TYPE AC_Unit_Status :
STRUCT
	bPresVal : BOOL;  // Stores ON/OFF state
    sUnitName : STRING;  // Stores unit name
END_STRUCT
END_TYPE

(* stored: Version 1.1.0.1, ProductVersion 3.1.4024.14
   DUT AC_Unit_Status: Id {5bfc5a03-a285-435e-add7-3e57241cc05e} *)
